// TIA Portal V19 export
DATA_BLOCK "DB_Panel_DP"   // DB86
{ S7_Optimized_Access := 'FALSE' }
AUTHOR : KHE_RE
NAME : DB_LADUN
VERSION : 2.0
// stored: AutoNumber false
   VAR RETAIN
      Anz_DP : Int := 8;   // * Anzahl Dosierpumpen
      Offset : Int := 20;   // * Beginn Daten
      Length : Int := 40;   // * Länge Daten
      res60 : Bool := FALSE;
      resB7 : Byte := 16#00;
      resB8 : Byte := 16#00;
      resB9 : Byte := 16#00;
      resB10 : Byte := 16#00;
      resB11 : Byte := 16#00;
      resD12 : DWord := 16#0000_0000;
      resD16 : DWord := 16#0000_0000;
      DoPu : Array[1..20] of Struct   // * Feldlänge anpassen
         Impulsdauer : Int;   // * Laufzeit Dosierimpuls [1/10 sec] (Falls keine Einstellmöglichkeit am PC)
         Impulspause : Int;   // * Pausenzeit zwischen zwei Impulsen [1/10 sec](Falls keine Einstellmöglichkeit
         resI : Int;
         Ein : Bool;   // Pumpe dauerhaft ein
         Auto : Bool;   // Pumpe Automatikbetrieb ein
         Kalibrierung : Bool;   // Pumpe in Kalibrierung
         res1 : Bool;
         res2 : Bool;
         Hand : Bool;   // Handdosierung läuft
         ON : Bool;   // DuPu läuft
         STM : Bool;   // DoPu Störung
         Kali_Start : Bool;   // Kalibrierung starten
         Kali_Stop : Bool;   // Kalibrierung anhalten
         res8 : Bool;
         res9 : Bool;
         res10 : Bool;
         res11 : Bool;
         res12 : Bool;
         res13 : Bool;
         Pumpleistung : Real;   // ml/s ml/Imp ....
         Zugabe_Hand : Real;   // ml
         Zugabe_Auto : Real;   // ml, ml/dm2
         RestDosierWert : Real;   // ml, Liter, g, kg usw.
         Kalibrierwert : Real;
         resD1 : DWord;
         resD2 : DWord;
         Kali_Count : DInt;   // Zählzelle Kalibrierdauer
      END_STRUCT;
   END_VAR
BEGIN
   DoPu[1..20].Impulsdauer := 1;
   DoPu[1..20].Impulspause := 1;
   DoPu[1..20].resI := 1;
   DoPu[1..20].Ein := FALSE;
   DoPu[1..4].Auto := TRUE;
   DoPu[5..20].Auto := FALSE;
   DoPu[1..20].Kalibrierung := FALSE;
   DoPu[1..20].res1 := FALSE;
   DoPu[1..20].res2 := FALSE;
   DoPu[1..20].Hand := FALSE;
   DoPu[1..20].ON := FALSE;
   DoPu[1..20].STM := FALSE;
   DoPu[1..20].Kali_Start := FALSE;
   DoPu[1..20].Kali_Stop := FALSE;
   DoPu[1..20].res8 := FALSE;
   DoPu[1..20].res9 := FALSE;
   DoPu[1..20].res10 := FALSE;
   DoPu[1..20].res11 := FALSE;
   DoPu[1..20].res12 := FALSE;
   DoPu[1..20].res13 := FALSE;
   DoPu[1..8].Pumpleistung := 0.1;
   DoPu[9..20].Pumpleistung := 0.0;
   DoPu[1..20].Zugabe_Hand := 0.0;
   DoPu[1..4].Zugabe_Auto := 10.0;
   DoPu[5..20].Zugabe_Auto := 0.0;
   DoPu[1].RestDosierWert := 0.0;
   DoPu[2].RestDosierWert := 0.09993901;
   DoPu[3..4].RestDosierWert := 0.09999623;
   DoPu[5..20].RestDosierWert := 0.0;
   DoPu[1..20].Kalibrierwert := 0.0;
   DoPu[1..20].resD1 := 16#0000_0000;
   DoPu[1..20].resD2 := 16#0000_0000;
   DoPu[1..20].Kali_Count := 0;
END_DATA_BLOCK
